FUNCTION_BLOCK Top
  (* Standard: 61499-2 *)
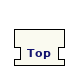
  FBS
    ticksource : Ticksource;
    gen1 : Generator;
    gen2 : Generator;
    ic1 : IntegralController;
    ic2 : IntegralController;
    load1 : Load;
    load2 : Load;
    tieline : Tieline;
    print : LfcPrint;
  END_FBS
  EVENT_CONNECTIONS
    ticksource.TickIc TO ic1.Tick;
    ticksource.TickIc TO ic2.Tick;
    ticksource.TickGen TO gen1.Tick;
    ticksource.TickGen TO gen2.Tick;
    ticksource.TickLoad TO load1.Tick;
    ticksource.TickLoad TO load2.Tick;
    ticksource.TickTie TO tieline.Tick;
    ticksource.TickPrint TO print.Tick;
    ic1.DprefChange TO print.DprefChange;
    ic2.DprefChange TO print.DprefChange;
    gen1.DfChange TO print.DfChange;
    gen2.DfChange TO print.DfChange;
    tieline.Dp12Change TO print.Dp12Change;
    ic1.DprefChange TO gen1.DprefChange;
    load1.DpeChange TO gen1.DpeChange;
    gen1.DfChange TO ic1.DfChange;
    tieline.Dp12Change TO ic1.Dp12Change;
    tieline.Dp12Change TO load1.Dp12Change;
    0 TO load1.DpeExternalChange;
    ic2.DprefChange TO gen2.DprefChange;
    load2.DpeChange TO gen2.DpeChange;
    gen2.DfChange TO ic2.DfChange;
    tieline.Dp12Change TO ic2.Dp12Change;
    tieline.Dp12Change TO load2.Dp12Change;
    0 TO load2.DpeExternalChange;
    gen1.DfChange TO tieline.DfChange;
    gen2.DfChange TO tieline.DfChange;
  END_CONNECTIONS
  DATA_CONNECTIONS
    ic1.Dpref TO print.Dpref1;
    ic2.Dpref TO print.Dpref2;
    gen1.Df TO print.Df1;
    gen2.Df TO print.Df2;
    tieline.Dp12 TO print.Dp12;
    ic1.Dpref TO gen1.Dpref;
    load1.Dpe TO gen1.Dpe;
    gen1.Df TO ic1.Df;
    tieline.Dp12 TO ic1.Dp12;
    tieline.Dp12 TO load1.Dp12;
    0 TO load1.DpeExternal;
    ic2.Dpref TO gen2.Dpref;
    load2.Dpe TO gen2.Dpe;
    gen2.Df TO ic2.Df;
    tieline.Dp21 TO ic2.Dp12;
    tieline.Dp21 TO load2.Dp12;
    0.1 TO load2.DpeExternal;
    gen1.Df TO tieline.Df1;
    gen2.Df TO tieline.Df2;
  END_CONNECTIONS
END_FUNCTION_BLOCK
